TYPE ST_Recipe_UCF_PARAM :
STRUCT
		//Sorter nasadek, typ produktu	
	iCapSorterProductType										:	ST_DIParametrr;		//:= 2; 		//		Typ produktu: 0- kule/fliptopy, 1- pompki, 2- disctop, 3-airless, 4-decoration cap (wyłączone podcisnienie na załapywarce), 5- decoration cap with new gripper (wyłączone podcisnienie + nowy program do robota)
	uiCapSorterIndexShow										:	ST_UdiParametr;	//:= 5;		//		Index produktu	
	bPresenceBottleEnableShow									:	ST_BoolParametr;					//		Sprawdzanie butelki w formatce

//--------------------------------------CapSorterTransporter-----------------------------------------------------------------------------------------------------------------------------	
	// Sorter nasadek, transporter zasobnika
	bCapSorterTransporterEnableShow								:	ST_BoolParametr;				//		Aktywacja
	iCapSorterTransporterTankConveyorVelocityShow				:	ST_DIParametrr;		//:= 1200;	//		Prędkość 							| [%] (1.0-100.0)
	iCapSorterTransporterStartDelayTimeShow						:	ST_DIParametrr;		//:= 100;		//		Timer do załączania 				| [ms] (0.0-10_000.0)
	udiCapSorterTransporterTimeProductOnSensorBeforeBrushShow	:	ST_UdiParametr;		//:= 150;		//		Timer pracy							| [ms] (0.0-10_000.0)
	iCapSorterTransporterEmptyingConveyorSpeedShow				:	ST_DIParametrr;		//:= 25;		// 		Prędkość, opróżnianie 				| [%] (1.0-100.0)
	iCapSorterTransporterVolumeOfCapsShow						:	ST_DIParametrr;		//:= 330;		//		Odłegłość do zamknięć, ostrzeżenie 	| [mm] (0.0-10_000.0)

//---------------------------------------CapSorterWheel----------------------------------------------------------------------------------------------------------------------------	
	// Sorter nasadek, stól
	bCapSorterWheelEnableShow									:	ST_BoolParametr;				//		Aktywacja
	lrCapSorterWheelMoveAccelerationEmptyTableShow				:   ST_LrParametr;			//:= 5000;	//		Dynamika rozpędzania - pusty 		| [obr/min²], (1.0-100_000.0) 
	lrCapSorterWheelMoveDecelerationEmptyTableShow				:   ST_LrParametr;			//:= 5000;    //		Dynamika spowalniania - pusty 		| [obr/min²] (1.0-100_000.0) 
	lrCapSorterWheelMoveSpeedEmptyTableShow						:   ST_LrParametr;		//:= 334;     //		Prędkość - pusty 					| [obr/min] (1.0-10_000.0)                
	lrCapSorterWheelMoveAngleEmptyTableShow						:   ST_LrParametr;			//:= 20;      //		Kąt - pusty 						| [obr/min] (0.0-360.0)                        
	lrCapSorterWheelJerkAngleEmptyTableShow						:   ST_LrParametr;		//:= 15000;   //		Zryw - pusty 						| [obr/min³] (1.0-1_000_000)                  
	iCapSorterWheelWaitingAfterRotationEmptyTableShow			:	ST_DIParametrr;		//:= 100;     //		Czas stabilizacji - pusty 			| [ms] (0.0-1_000)                 
	                                                                        //
	lrCapSorterWheelMoveAccelerationFullTableShow				:   ST_LrParametr;		//:= 5000;	//		Dynamika rozpędzania - pełny 		| [obr/min²], (1.0-100_000.0) 
	lrCapSorterWheelMoveDecelerationFullTableShow				:   ST_LrParametr;		//:= 5000;    //		Dynamika spowalniania - pełny 		| [obr/min²] (1.0-100_000.0) 
	lrCapSorterWheelMoveSpeedFullTableShow						:   ST_LrParametr;		//:= 334;     //		Prędkość - pełny 					| [obr/min] (1.0-10_000.0)                
	lrCapSorterWheelMoveAngleFullyTableShow						:   ST_LrParametr;			//:= 6;       //		Kąt - pełny 						| [obr/min] (0.0-360.0)                        
	lrCapSorterWheelJerkAngleFullTableShow						:   ST_LrParametr;			//:= 15000;   //		Zryw - pełny 						| [obr/min³] (1.0-1_000_000)                  
	iCapSorterWheelWaitingAfterRotationFullTableShow			:	ST_DIParametrr;		//:= 30;      //		Czas stabilizacji - pełny 			| [ms] (0.0-1_000)                 
	                                                                        //
	lrCapSorterWheelMoveAccelerationHalfFullTableShow			:   ST_LrParametr;			//:= 5000;	//		Dynamika rozpędzania - półpełny 	| [obr/min²], (1.0-100_000.0) 
	lrCapSorterWheelMoveDecelerationHalfFullTableShow			:   ST_LrParametr;			//:= 5000;    //		Dynamika spowalniania - półpełny 	| [obr/min²] (1.0-100_000.0) 
	lrCapSorterWheelMoveSpeedHalfFullTableShow					:   ST_LrParametr;			//:= 334;     //		Prędkość - półpełny 				| [obr/min] (1.0-10_000.0)                
	lrCapSorterWheelMoveAngleHalfFullyTableShow					:   ST_LrParametr;			//:= 12;      //		Kąt - półpełny						| [obr/min] (0.0-360.0)                        
	lrCapSorterWheelJerkAngleHalfFullTableShow					:   ST_LrParametr;			//:= 15000;   //		Zryw - półpełny 					| [obr/min³] (1.0-1_000_000)                  
	iCapSorterWheelWaitingAfterRotationHalfFullTableShow		:	ST_DIParametrr;		//:= 50;      //		Czas stabilizacji - półpełny 		| [ms] (0.0-1_000)                 

//-------------------------------------CapSorterCamera------------------------------------------------------------------------------------------------------------------------------	                                                    	
	// Sorter nasadek, system wizyjny
	
    bCapSorterCameraEnableShow									:	ST_BoolParametr;				//	[H]	Aktywacja                            	
	
//-----------------------------------------CapSorterRobot--------------------------------------------------------------------------------------------------------------------------	
	// Sorter nasadek, robot
	bCapSorterRobotEnableShow									:	ST_BoolParametr;				//		Aktywacja
                                                                                                                           	
	lrCapSorterRobotPlace1PositionXShow							:   ST_LrParametr;					//		Offset odkładania 1, X 			| [mm]	((-100.0)-100.0)       
	lrCapSorterRobotPlace1PositionYShow							:   ST_LrParametr;	    			//		Offset odkładania 1, Y 			| [mm]	((-100.0)-100.0)       
	lrCapSorterRobotPlace1PositionZShow							:   ST_LrParametr;	    			//		Offset odkładania 1, Z 			| [mm]	((-100.0)-100.0)       
	lrCapSorterRobotPlace1PositionCShow							:   ST_LrParametr;	    			//		Offset odkładania 1, C 			| [° ]	((-360.0)-360.0)                 
	iCapSorterRobotPickElevationShow							:	ST_DIParametrr;				//		Punkt nad poz. Pick				| [mm]	(30-1000)
	iCapSorterRobotPickTimeShow									:	ST_DIParametrr;					//		Czas przyssania					| [ms]	(0-10_000)
	iCapSorterRobotVacuumActivationShow							:	ST_DIParametrr;					//		Czas przed przyssaniem			| [ms]	(0-1000)
	iCapSorterRobotVacuumOffShow								:	ST_DIParametrr;					//		Czas przed oddmuchem			| [ms]	(0-1000)
	iCapSorterRobotPlaceTimeShow								:	ST_DIParametrr;					//		Czas oddmuchu					| [ms]	(0-1000)
	iCapSorterRobotTCP_PlaceOffsetShow							:	ST_DIParametrr;					//		Wysokość od TCP do p. odłożenia	| [mm]	(0-1000)									
	iCapSorterRobotAccelerationDecelerationShow					:	ST_DIParametrr;					//		Dynamika rozpędzania/hamowania	| [%]	(20-100)
	iCapSorterRobotGripperWatchdogShow							:	ST_DIParametrr;					//		Czas sprawdzania silownika		| [ms]	(0-1000)
	iCapSorterRobotParalaxCorrectionShow						:	ST_DIParametrr;				//		Korekta paralaxy				| [mm]	(0-100)
	
	iCapSorterRobotNumberToolShow								:	ST_DIParametrr;				//		Numer narzędzia					| 		(0-10)
	iCapSorterRobotPickPositionZShow							:	ST_DIParametrr;					//		Wysokość pobierania 			| [mm]	(0-200)
	iCapSorterRobotTCP_Lenght									:	ST_DIParametrr;					//		Długość chwytaka				| [mm]	(10-100)
	iCapSorterRobotProductDiametr								:	ST_DIParametrr;					//		Średnica nasadki				| [mm] 	(10-100)
	
//----------------------------------------CapSorterIntermediateTransporter---------------------------------------------------------------------------------------------------------------------------
	// Sorter nasadek, transporter zasypowy
	bCapSorterIntermediateTransporterEnableShow					:	ST_BoolParametr;			//		Aktywacja
	iCapSorterIntermediateTransporterAutoSpeedShow				:	ST_DIParametrr;		//:= 20;		//		Prędkość 					| [%] (1.0-100.0)
	iCapSorterIntermediateTransporterManualSpeedShow			:	ST_DIParametrr;		//:= 30;		//		Prędkość, manual 			| [%] (1.0-100.0)
	iCapSorterIntermediateTransporterEmptyingSpeedShow			:	ST_DIParametrr;		//:= 50;		//		Prędkość, opróżnianie 		| [%] (1.0-100.0)
	iCapSorterIntermediateTransporterDelayCountTimeShow			:	ST_DIParametrr;		//:= 100;		//		Timer pracy					| [ms]	(0.0-100_000.0)
	iCapSorterIntermediateTransporterReverseTimeShow			:	ST_DIParametrr;		//:= 4000;	//		Timer odwróconej pracy 		| [ms] (0.0-10_000.0)
	udiCapSorterIntermediateTransporterTimeProductOnSensorShow	:	ST_UdiParametr;		//:= 1800;	//		Czas produktu na czujniku 	| [ms] (0.0-10_000.0)	
	lrCapSorterIntermediateTransporterWheelAngleShow			:   ST_LrParametr;			//:= 6;		//		Kąt zasypu 					| [°] (1.0-360.0)
	
//----------------------------------------CapSorterIntermediateBrush---------------------------------------------------------------------------------------------------------------------------
	//Sorter nasadek, szczotka transportera
	bCapSorterIntermediateBrushEnableShow						:	ST_BoolParametr;				//		Aktywacja
	iCapSorterIntermediateBrushAutoSpeedShow					:	ST_DIParametrr;		//:= 30;		//		Prędkość  					| [%] (0.0-100.0)
	iCapSorterIntermediateBrushManualSpeedShow					:	ST_DIParametrr;		//:= 30;		//		Prędkość, manual 			| [%] (0.0-100.0)
	iCapSorterIntermediateBrushEmptyingSpeedShow				:	ST_DIParametrr;		//:= 30;		//		Prędkość, opróżnianie 		| [%] (0.0-100.0)
	lrCapSorterIntermediateBrushPositionHeightSVShow			:   ST_LrParametr;			//:= 45;		//		Wysokość 					| [mm] (0.0-10_000.0)

//----------------------------------------CapSorterBrush1OnWheel---------------------------------------------------------------------------------------------------------------------------
	// Sorter nasadek, szczotka stolu 1
	bCapSorterBrush1OnWheelEnableShow							:	ST_BoolParametr;					//		Aktywacja
	iCapSorterBrush1OnWheelAutoSpeedShow						:	ST_DIParametrr;		//:= 30;		//		Prędkość 					| [%] (0.0-100.0)
	iCapSorterBrush1OnWheelManualSpeedShow						:	ST_DIParametrr;		//:= 30;		//		Prędkość, manual 			| [%] (0.0-100.0)
	iCapSorterBrush1OnWheelEmptyingSpeedShow					:	ST_DIParametrr;		//:= 30;		//		Prędkość, opróżnianie 		| [%] (0.0-100.0)
	lrCapSorterBrush1OnWheelPositionHeightSVShow				:   ST_LrParametr;			//:= 45;		//		Wysokość 					| [mm] (0.0-10_000.0)
	
//----------------------------------------CapSorterBrush2OnWheel----------------------------------------------------------------------------------
	// Sorter nasadek, szczotka stolu 2
	bCapSorterBrush2OnWheelEnableShow							:	ST_BoolParametr;					//		Aktywacja
	iCapSorterBrush2OnWheelAutoSpeedShow						:	ST_DIParametrr;		//:= 30;		//		Prędkość 					| [%] (0.0-100.0)
	iCapSorterBrush2OnWheelManualSpeedShow						:	ST_DIParametrr;		//:= 30;		//		Prędkość, manual 			| [%] (0.0-100.0)
	iCapSorterBrush2OnWheelEmptyingSpeedShow					:	ST_DIParametrr;		//:= 30;		//		Prędkość, opróżnianie 		| [%] (0.0-100.0)
	lrCapSorterBrush2OnWheelPositionHeightSVShow				:   ST_LrParametr;		//:= 45;		//		Wysokość 					| [mm] (0.0-10_000.0)

//------------------------------------------CapFeeder-------------------------------------------------------------------------------------------------------------------------	
	// Sorter nasadek, 
	bCapSorterFeederEnableShow									:	ST_BoolParametr;				//		Aktywacjaa
	bCapSorterFeederEnableTubeError								:	ST_BoolParametr;				// 		Aktywacja błedu słomki
	lrCapSorterFeederMover1InputPositionShow					:   ST_LrParametr;					//		Pozycja wkładania, wózek 1 	| [mm] (?-?)
	lrCapSorterFeederMover2InputPositionShow					:   ST_LrParametr;					//		Pozycja wkładania, wózek 2 	| [mm] (?-?)
	lrCapSorterFeederMover1OutputPositionShow					:   ST_LrParametr;					//		Pozycja wyjmowania, wózek 1 | [mm] (?-?)
	lrCapSorterFeederMover2OutputPositionShow					:   ST_LrParametr;					//		Pozycja wyjmowania, wózek 2 | [mm] (?-?)
	lrCapSorterFeederSlotDistanceShow							:   ST_LrParametr;					//		Offset wkładania			| [mm] (?-?)			Old-(Odstęp między pozycjami kładzenia)
	lrCapSorterFeederMoverSpeedShow								:   ST_LrParametr;					//		Prędkość				 	| [%] (0.0-100.0)
	lrCapSorterFeederMoverAccelerationShow						:   ST_LrParametr;					//		Przyspieszenie 				| [mm/s²] 
	lrCapSorterFeederMoveJerkShow								:   ST_LrParametr;				//		Zryw						| [mm/s³]

//-------------------------------------------------------------------------------------------------------------------------------------------------------------------	
	//CapPreScrewer		
	bCapSorterPreScrewerEnableShow								:	ST_BoolParametr;				// 		Aktywacja
	bCapSorterPreScrewerPicker1EnableShow						:	ST_BoolParametr;			// 		Aktywacja	
	bCapSorterPreScrewerPicker2EnableShow						:	ST_BoolParametr;			// 		Aktywacja
	bCapSorterPreScrewerPicker3EnableShow						:	ST_BoolParametr;				// 		Aktywacja	
	bCapSorterPreScrewerPicker4EnableShow						:	ST_BoolParametr;				// 		Aktywacja
	//Oś Z
	lrCapSorterPreScrewerPickZPositionShow						:   ST_LrParametr;					//		Wysokość pobierania						| [mm]	
	lrCapSorterPreScrewerCatcherReleseShow						:   ST_LrParametr;					//		nie używamy Wysokość otwierania chwytaka nakrętek	| [mm]		
	lrCapSorterPreScrewerCapCatcherZPositionShow				:   ST_LrParametr;					//		Wysokość zamykania nakrętkek			| [mm]
	lrCapSorterPreScrewerTopZPositionShow						:   ST_LrParametr;					//		Pozycja górna ośi Z						| [mm] 	
	lrCapSorterPreScrewerCartesianCatchZPositionShow			:   ST_LrParametr;	 				//      Wait Position
	lrCapSorterPreScrewerStrawCatcherZPositionShow				:   ST_LrParametr;					//		Wysokość otwierania łapaczy słomek		| [mm]	
	LrCapSorterPreScrewerCheckStrawCatcherActuatorZPosition		:   ST_LrParametr;					//		Wysokość sparawdzania cofania łapaczy słomek	| [mm]	
	lrCapSorterPreScrewerScrewerStartZPositionShow				:   ST_LrParametr;					//		Wysokość początku zakręcania			| [mm]	
	lrCapSorterPreScrewerGripperOpenPositionShow				:   ST_LrParametr;					//		Pozycja otwierania chwytaka butelek 	| [mm]
	lrCapSorterPreScrewerPlaceZPositionShow						:   ST_LrParametr;					//		Wysokość odkładania - koniec załapywania gwintu	| [mm]   	
	//Wspólne ruchi	
	lrCapSorterPreScrewerBendingDistanceShow					:   ST_LrParametr;					//		Odległość zaokrąglania ruchów 			| [mm]		
	lrCapSorterPreScrewerStrawInsertDistance					:   ST_LrParametr;					//		Odległość wspólnego ruchu, prowadzenie słomki	| [mm]		
	//Oś x
	lrCapSorterPreScrewerPickXMover1PositionShow				:   ST_LrParametr;				//		Pozycja osi poziomej do pobierania, wozek 1	| [mm]
	lrCapSorterPreScrewerPickXMover2PositionShow				:   ST_LrParametr;					//		Pozycja osi poziomej do pobierania, wozek 2	| [mm]
	lrCapSorterPreScrewerPlaceXPositionShow						:   ST_LrParametr;			//		Pozycja osi poziomej do odkładania			| [mm]
	//Oś zakręcania
	lrCapSorterPreScrewerScrewFindingShow						:   ST_LrParametr;					//		Kąt szukania gwintu							| [°]
	lrCapSorterPreScrewerScrewDistanceShow						:   ST_LrParametr;					//		Kąt zakręcania								| [°]
	//Prédkośći                                                                                                                         	
	lrCapSorterPreScrewerPickerSpeedShow						:   ST_LrParametr;					//		Prędkość									| [mm/s]   
	lrCapSorterPreScrewerPickerAccelerationShow					:   ST_LrParametr;				//		Przyspieszenie								| [mm/s²] 		
	lrCapSorterPreScrewerPickerJerkShow							:   ST_LrParametr;					//		Zryw										| [mm/s³]
                                                                                                                                        	
	lrCapSorterPreScrewerCatcherSpeedShow						:   ST_LrParametr;					//		Prędkość									| [mm/s] 
	lrCapSorterPreScrewerCatcherAccelerationShow				:   ST_LrParametr;					//		Przyspieszenie								| [mm/s²] 	
	lrCapSorterPreScrewerCatcherJerkShow						:   ST_LrParametr;					//		Zryw										| [mm/s³]	                                                                                                                                 	
	lrCapSorterPreScrewerScrewSpeedShow							:   ST_LrParametr;					//		Prędkość zakręcania							| [mm/s]
	lrCapSorterPreScrewerScrewAccelerationShow					:   ST_LrParametr;					//		Przyspieszenie zakręcania				| [mm/s²]
	lrCapSorterPreScrewerScrewJerkShow							:   ST_LrParametr;				//		Zryw zakręcania							| [mm/s³]

	//Oś łapacza słomki	
	lrCapSorterPreScrewerCatcherCatchingPositionShow			:   ST_LrParametr;					//		Pozycja łapania słomki					| [mm]
	lrCapSorterPreScrewerCatcherPlacePositionShow				:   ST_LrParametr;					//		Pozycja dolna łapacza słomki			| [mm]
	lrCapSorterPreScrewerCatcherHightSVShow						:   ST_LrParametr;					//		Nastawa wysokości stacji łapacza słomek		| [mm]
	//Kalibracja chwytaków butelki
	bCapSorterPreScrewerBottleCatcherEnableShow					:	ST_BoolParametr;			//		Actywacja chwytaków butelki
	lrCapSorterPreScrewerBottleCatch1OpenValueShow				:   ST_LrParametr;					//		Chwytak 1 | wartość kalibracji otwartego chwytaka
	lrCapSorterPreScrewerBottleCatch1CloseValueShow				:   ST_LrParametr;					//		Chwytak 1 | wartośc kalibracji zamkniętego chwytaka
	lrCapSorterPreScrewerBottleCatch2OpenValueShow				:   ST_LrParametr;					//		Chwytak 2 | wartość kalibracji otwartego chwytaka
	lrCapSorterPreScrewerBottleCatch2CloseValueShow				:   ST_LrParametr;					//		Chwytak 2 | wartość kalibracji zamkniętego chwytaka
	lrCapSorterPreScrewerBottleCatch3OpenValueShow				:   ST_LrParametr;	                //		Chwytak 3 | wartość kalibracji otwartego chwytaka
	lrCapSorterPreScrewerBottleCatch3CloseValueShow				:   ST_LrParametr;					//		Chwytak 3 | wartość kalibracji zamkniętego chwytaka	
	lrCapSorterPreScrewerBottleCatch4OpenValueShow				:   ST_LrParametr;	                //		Chwytak 4 | wartość kalibracji otwartego chwytaka
	lrCapSorterPreScrewerBottleCatch4CloseValueShow				:   ST_LrParametr;					//		Chwytak 4 | wartość kalibracji zamkniętego chwytaka
	                                                        	
	lrCapSorterPreScrewerBottleCatchToleranceValueShow			:   ST_LrParametr;				//		Tolerancja chwytaków
	lrCapSorterPreScrewerCatchAngleOpenSV						:   ST_LrParametr;		//:= 180.0;		//		[] Kąt puszczania centrowników
	
	lrCapSorterPreScrewerWaitInPlaceTimeShow					:   ST_LrParametr;		//:= 50;			//		Czas zatrzymania w miejscu odłożenia 	| [ms]
	
	bCapSorterPreScrewerCatchAngleOpenEnaShow					:	ST_BoolParametr;					// 		Aktywacja puszczania centrowników po osiągnięciu zadanego kątu
	bCapSorterPreScrewerPoundedInCap							:	ST_BoolParametr;				// 		Wbijana nasadka
	
//Parametry do obliczeń 
	lrCapSorterBottleHightShow									:   ST_LrParametr;					//		Wysokość butelki
	lrCapSorterBottleNeckHightShow								:   ST_LrParametr;					// 		Wysokość szyjki butelki
	lrCapSorterCapHightShow										:   ST_LrParametr;					// 		Wysokość zamknięcia
	lrCapSorterCapNeckHightShow									:   ST_LrParametr;					//		Wysokość szyjki zamknięcia

//Rezerwa	
	lrCapSorterSpare1											:   ST_LrParametr;					//Rezerwa 1
	lrCapSorterSpare2											:   ST_LrParametr;					//Rezerwa 2
	lrCapSorterSpare3											:   ST_LrParametr;					//Rezerwa 3
	lrCapSorterSpare4											:   ST_LrParametr;					//Rezerwa 4
	lrCapSorterSpare5											:   ST_LrParametr;					//Rezerwa 5
	lrCapSorterSpare6											:   ST_LrParametr;					//Rezerwa 6
	lrCapSorterSpare7											:   ST_LrParametr;					//Rezerwa 7	


	lrCapSorterPreScrewerPickerSpeedWhenScrewerShow				:	ST_LrParametr;

END_STRUCT
END_TYPE

(* stored: Version 1.2.0.0, ProductVersion 3.1.4026.13, FileIdentifier f5009a2eaf86076281deb777078524f1efd40c7d, FileSignature 135c7cfcd48df1ef1b25cc92aa8f6872dee66904d935c2f91d3345b8e8ef9c673049b10bf9d2f9ffff063e0b4aedf46eade0b6f5eeac05dfcc61221f3e67be955ab8f241e075ba9ad0e2990f76faecbc8199eb6b1088f89c4a0c29e3dff7eba4c76455c70da5e409bda19f2649bcefaf1d1a23be9424b301388b02e79783925550fd0617e5a38d90683461cf3dcecf260dba77d956180bfeba59ba499f174a5bc3079bd6cf7caf15884b080cae8a1c5faceb9e9cd295c634b3436931bcf319cf178e0d4eff43445e1730d16e1a434c5905fb180c9b83aee5bb5cf28d43bd4e008badf013e5079ad1594b1735e87689f826f0d40adb769a1668821ab49f4cc6a4
   DUT ST_Recipe_UCF_PARAM: Id {1e035f46-353e-4776-a4eb-d1df67b060ec} *)
